(* PLC project Unnamed, Unknown Unnamed 1 *)
(* stored: creationDateTime 2025-11-05T10:04:27, modificationDateTime 2025-11-05T10:11:24 *)

PROGRAM main
  VAR
    I_PushButton : BOOL := False;
    PB_Down : BOOL := False;
    PB_Up : BOOL := False;
  END_VAR

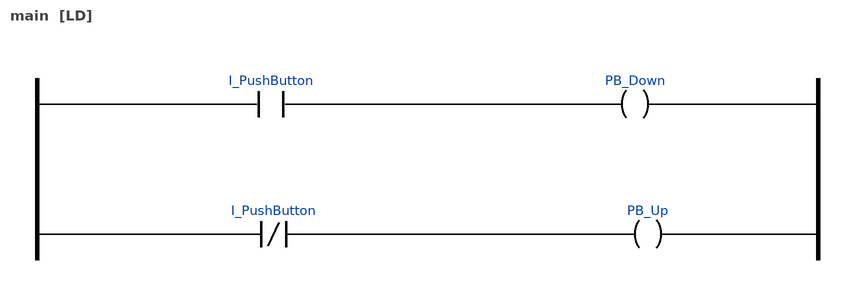
(* LD diagram, written out as Structured Text *)
PB_Down := I_PushButton;
PB_Up := NOT I_PushButton;
END_PROGRAM

CONFIGURATION Config0
  RESOURCE Res0 ON PLC
    TASK task0(INTERVAL := T#20ms, PRIORITY := 0);
    PROGRAM instance0 WITH task0 : main;
  END_RESOURCE
END_CONFIGURATION
